FUNCTION_BLOCK SS5_ifb_ps_Camera (* nn *)
  (* Standard: 61499-2 *)
  (* Version 1.0, 2025-07-23, PS_Transformer_for_Unknown *)
  PACKAGE UserLibs::SubStations::SS5;
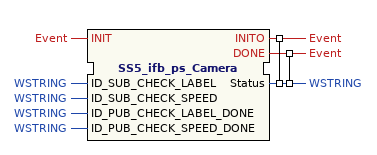
  EVENT_INPUT
    INIT;
  END_EVENT
  EVENT_OUTPUT
    INITO WITH Status;
    DONE WITH Status;
  END_EVENT
  VAR_INPUT
    ID_SUB_CHECK_LABEL : WSTRING;
    ID_SUB_CHECK_SPEED : WSTRING;
    ID_PUB_CHECK_LABEL_DONE : WSTRING;
    ID_PUB_CHECK_SPEED_DONE : WSTRING;
  END_VAR
  VAR_OUTPUT
    Status : WSTRING;
  END_VAR
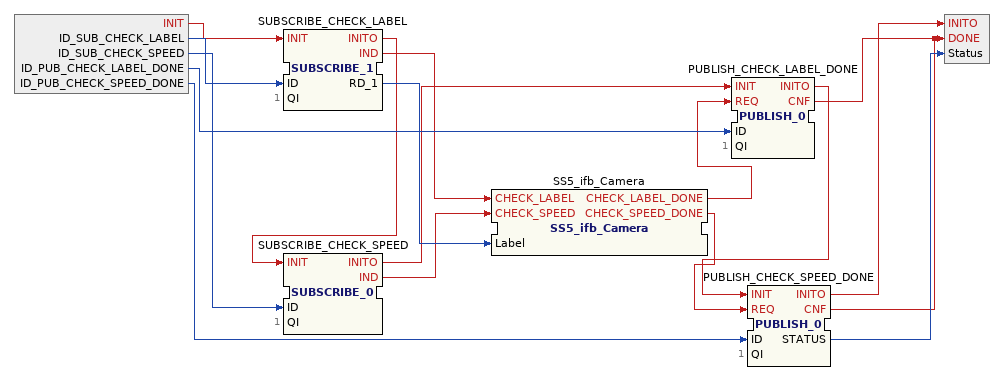
  FBS
    SUBSCRIBE_CHECK_LABEL : SUBSCRIBE_1(QI := 1);
    SUBSCRIBE_CHECK_SPEED : SUBSCRIBE_0(QI := 1);
    PUBLISH_CHECK_LABEL_DONE : PUBLISH_0(QI := 1);
    PUBLISH_CHECK_SPEED_DONE : PUBLISH_0(QI := 1);
    SS5_ifb_Camera : UserLibs::SubStations::SS5::SS5_ifb_Camera;
  END_FBS
  EVENT_CONNECTIONS
    INIT TO SUBSCRIBE_CHECK_LABEL.INIT;
    SUBSCRIBE_CHECK_LABEL.INITO TO SUBSCRIBE_CHECK_SPEED.INIT;
    SUBSCRIBE_CHECK_SPEED.INITO TO PUBLISH_CHECK_LABEL_DONE.INIT;
    PUBLISH_CHECK_LABEL_DONE.INITO TO PUBLISH_CHECK_SPEED_DONE.INIT;
    PUBLISH_CHECK_SPEED_DONE.INITO TO INITO;
    PUBLISH_CHECK_LABEL_DONE.CNF TO DONE;
    PUBLISH_CHECK_SPEED_DONE.CNF TO DONE;
    SUBSCRIBE_CHECK_LABEL.IND TO SS5_ifb_Camera.CHECK_LABEL;
    SUBSCRIBE_CHECK_SPEED.IND TO SS5_ifb_Camera.CHECK_SPEED;
    SS5_ifb_Camera.CHECK_LABEL_DONE TO PUBLISH_CHECK_LABEL_DONE.REQ;
    SS5_ifb_Camera.CHECK_SPEED_DONE TO PUBLISH_CHECK_SPEED_DONE.REQ;
  END_CONNECTIONS
  DATA_CONNECTIONS
    ID_SUB_CHECK_LABEL TO SUBSCRIBE_CHECK_LABEL.ID;
    ID_SUB_CHECK_SPEED TO SUBSCRIBE_CHECK_SPEED.ID;
    ID_PUB_CHECK_LABEL_DONE TO PUBLISH_CHECK_LABEL_DONE.ID;
    ID_PUB_CHECK_SPEED_DONE TO PUBLISH_CHECK_SPEED_DONE.ID;
    SUBSCRIBE_CHECK_LABEL.RD_1 TO SS5_ifb_Camera.Label;
    PUBLISH_CHECK_SPEED_DONE.STATUS TO Status;
  END_CONNECTIONS
END_FUNCTION_BLOCK
